FUNCTION_BLOCK Recipe_10051_Proberezept
VAR_INPUT
	execute	: BOOL;
	Order	: DUT_RECIPEORDER;
END_VAR
VAR_OUTPUT
	RecipeInfo	: DUT_RECIPEOFFER;
	RecipeDone	: BOOL;	
	InitDone	: BOOL;
END_VAR
VAR
	StepDone	: BOOL;
END_VAR

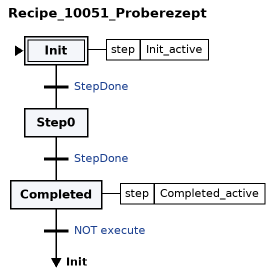
INITIAL_STEP Init:
    Init_active(N);  // step action
END_STEP
TRANSITION FROM Init TO Step0
    := StepDone;
END_TRANSITION
STEP Step0:
END_STEP
TRANSITION FROM Step0 TO Completed
    := StepDone;
END_TRANSITION
STEP Completed:
    Completed_active(N);  // step action
END_STEP
TRANSITION FROM Completed TO Init
    := NOT execute;
END_TRANSITION

ACTION Completed_active:
RecipeDone := TRUE;
StepDone := FALSE;
END_ACTION

ACTION Init_active:
RecipeDone := FALSE;

// Initialisation of Recipe Parameters an name etc
RecipeInfo.Name := 'Pump Test';
RecipeInfo.Description := 'Test of all 8 Pumps';
RecipeInfo.Dummy := FALSE;
RecipeInfo.RecipeID := 10050; 	// 
Initdone := TRUE;

//Parameter 0:
(*
	RecipeInfo.UserParameter[0].Dummy 		:= 
	RecipeInfo.UserParameter[0].Default		:=
	RecipeInfo.UserParameter[0].Description	:=
	RecipeInfo.UserParameter[0].MaxValue	:=
	RecipeInfo.UserParameter[0].MinValue	:=
	RecipeInfo.UserParameter[0].Name		:=
	RecipeInfo.UserParameter[0].Unit		:=
*)
//Parameter 1:
(*
	RecipeInfo.UserParameter[1].Dummy 		:= 
	RecipeInfo.UserParameter[1].Default		:=
	RecipeInfo.UserParameter[1].Description	:=
	RecipeInfo.UserParameter[1].MaxValue	:=
	RecipeInfo.UserParameter[1].MinValue	:=
	RecipeInfo.UserParameter[1].Name		:=
	RecipeInfo.UserParameter[1].Unit		:=
*)
//Parameter 2:

(*
	RecipeInfo.UserParameter[2].Dummy 		:= 
	RecipeInfo.UserParameter[2].Default		:=
	RecipeInfo.UserParameter[2].Description	:=
	RecipeInfo.UserParameter[2].MaxValue	:=
	RecipeInfo.UserParameter[2].MinValue	:=
	RecipeInfo.UserParameter[2].Name		:=
	RecipeInfo.UserParameter[2].Unit		:=
*)

//Parameter 3:

(*
	RecipeInfo.UserParameter[3].Dummy 		:= 
	RecipeInfo.UserParameter[3].Default		:=
	RecipeInfo.UserParameter[3].Description	:=
	RecipeInfo.UserParameter[3].MaxValue	:=
	RecipeInfo.UserParameter[3].MinValue	:=
	RecipeInfo.UserParameter[3].Name		:=
	RecipeInfo.UserParameter[3].Unit		:=
*)

//Parameter 4:

(*
	RecipeInfo.UserParameter[4].Dummy 		:= 
	RecipeInfo.UserParameter[4].Default		:=
	RecipeInfo.UserParameter[4].Description	:=
	RecipeInfo.UserParameter[4].MaxValue	:=
	RecipeInfo.UserParameter[4].MinValue	:=
	RecipeInfo.UserParameter[4].Name		:=
	RecipeInfo.UserParameter[4].Unit		:=
*)


//Parameter 5:

(*
	RecipeInfo.UserParameter[5].Dummy 		:= 
	RecipeInfo.UserParameter[5].Default		:=
	RecipeInfo.UserParameter[5].Description	:=
	RecipeInfo.UserParameter[5].MaxValue	:=
	RecipeInfo.UserParameter[5].MinValue	:=
	RecipeInfo.UserParameter[5].Name		:=
	RecipeInfo.UserParameter[5].Unit		:=
*)
END_ACTION

END_FUNCTION_BLOCK

(* stored: Version 1.1.0.1, ProductVersion 3.1.0.25
   POU Recipe_10051_Proberezept: Id {04ec139a-9327-4bd4-ba77-abe45aece90c}
   Action Completed_active: Id {25601c23-c991-4275-8f79-31de094e17b2}
   Action Init_active: Id {35646272-bddb-454a-8a50-b5351194028c} *)
